// TIA Portal V17 export
// export: Created 2024-01-30T08:49:16.1319613Z, ExportSetting WithDefaults, DisplayName Totally Integrated Automation Portal, DisplayVersion V17 Update 6, DisplayName TIA Portal Openness, DisplayVersion V17 Update 6, DisplayName TIA Portal Version Control Interface, DisplayVersion V17, DisplayName STEP 7 Professional, DisplayVersion V17 Update 6, DisplayName STEP 7 Safety, DisplayVersion V17 Update 6, DisplayName WinCC Advanced, DisplayVersion V17 Update 6
DATA_BLOCK "FB_DATA_LOGGING_DB"   // DB26
VERSION : 0.1
// stored: AutoNumber true, DBAccessibleFromOPCUA true, DBAccessibleFromWebserver true, InstanceOfName FB_DATA_LOGGING, InstanceOfType FB
"FB_DATA_LOGGING"
   // VAR
   //    DataLogCreate_Instance { S7_SetPoint := 'True'} : DataLogCreate;
   //    DataLogWrite_Instance { S7_SetPoint := 'True'} : DataLogWrite;
   //    DataLogNewFile_Instance { S7_SetPoint := 'True'} : DataLogNewFile;
   //    DataLogNewFile_Instance_1 { S7_SetPoint := 'True'} : DataLogNewFile;
   //    DataLogDelete_Instance { S7_SetPoint := 'True'} : DataLogDelete;
   //    DataLogClear_Instance { S7_SetPoint := 'True'} : DataLogClear;
   // END_VAR
BEGIN
END_DATA_BLOCK
